// TIA Portal V17 export
// export: Created 2023-05-07T12:12:24.5179636Z, ExportSetting WithDefaults, DisplayName Totally Integrated Automation Portal, DisplayVersion V17, DisplayName TIA Portal Openness, DisplayVersion V17, DisplayName TIA Portal Version Control Interface, DisplayVersion V17, DisplayName TIA Portal Test Suite Advanced, DisplayVersion V17, DisplayName STEP 7 Professional, DisplayVersion V17, DisplayName SIMATIC Energy Suite, DisplayVersion V17, DisplayName STEP 7 Safety, DisplayVersion V17, DisplayName WinCC Professional, DisplayVersion V17
VAR_GLOBAL   // PLC tag table "Input"
   I_LevelMeter AT %ID30 : Real;
   I_FlowMeter AT %ID34 : Real;
   I_FactoryRuning AT %I0.0 : Bool;
END_VAR
